FUNCTION_BLOCK Button_HMI (* Service Interface Function Block Type *)
  (* Standard: 61499-2 *)
  (* Version 0.0, 5/25/2016, Andrei, nxtControl GmbH, template *)
  PACKAGE Main;
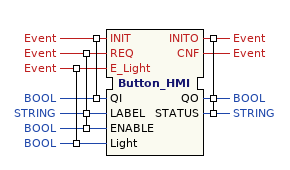
  EVENT_INPUT
    INIT WITH QI;
    REQ WITH LABEL, ENABLE;
    E_Light WITH Light;
  END_EVENT
  EVENT_OUTPUT
    INITO WITH QO, STATUS;
    CNF;
  END_EVENT
  VAR_INPUT
    QI : BOOL;
    LABEL : STRING;
    ENABLE : BOOL;
    Light : BOOL;
  END_VAR
  VAR_OUTPUT
    QO : BOOL; (* Event Output Qualifier *)
    STATUS : STRING; (* Service Status *)
  END_VAR
  SERVICE /
    SEQUENCE 
    END_SEQUENCE
  END_SERVICE
END_FUNCTION_BLOCK
